FUNCTION proj7_TupleStruct_1: REAL
{ S7_Optimized_Access := 'false' }
    VAR_INPUT
        tuple: TupleStruct_1;
    END_VAR

BEGIN
    proj7_TupleStruct_1 := tuple.field7;
END_FUNCTION
